FUNCTION_BLOCK ArucoDetector (* openCV Aruco Detector *)
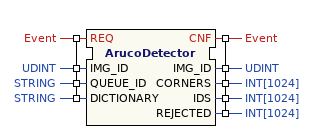
  EVENT_INPUT
    REQ WITH IMG_ID, QUEUE_ID, DICTIONARY;
  END_EVENT
  EVENT_OUTPUT
    CNF WITH IMG_ID, CORNERS, IDS, REJECTED;
  END_EVENT
  VAR_INPUT
    IMG_ID : UDINT;
    QUEUE_ID : STRING;
    DICTIONARY : STRING;
  END_VAR
  VAR_OUTPUT
    IMG_ID : UDINT;
    CORNERS : ARRAY [0..1023] OF INT;
    IDS : ARRAY [0..1023] OF INT;
    REJECTED : ARRAY [0..1023] OF INT;
  END_VAR
END_FUNCTION_BLOCK
